PROGRAM prgLab16
VAR
	rAddSin:LREAL:=0.01;
	rResultSin:LREAL;
	rSin:LREAL;
	rAddTri:LREAL:=0.01;
	rResultTri:LREAL:=0.01;
	rTri:LREAL;
	rVector:ARRAY[1..5] OF LREAL:=[1,5,6,2,8];
END_VAR

rResultSin:=rResultSin+rAddSin;
rSin:=SIN(rResultSin);

rTri:=rTri+rResultTri;
IF rTri>=1 THEN
	rResultTri:= -rAddTri;
ELSIF rTri <=-1 THEN
	rResultTri:= rAddTri;
END_IF

END_PROGRAM

(* stored: Version 1.1.0.1, ProductVersion 3.1.4024.11
   POU prgLab16: Id {b2de806b-72e7-491e-8489-90d0479cacb9}, SpecialFunc None *)
